{attribute 'linkalways'} 
{attribute 'no_explicit_call' := 'This FB is a CLASS and must be accessed using methods or properties'}
{attribute 'enable_dynamic_creation'}
FUNCTION_BLOCK FINAL MAX_UDINT EXTENDS Node
VAR
	in1 : _UDINT(0);
	in2 : _UDINT(0);
	out : _UDINT(0);
END_VAR

METHOD PUBLIC Clone : I_Node
VAR
	pNode : POINTER TO MAX_UDINT;
END_VAR
pNode := __NEW(MAX_UDINT);
Clone := pNode^;
END_METHOD

METHOD FB_init : BOOL
VAR_INPUT
	bInitRetains : BOOL; // if TRUE, the retain variables are initialized (warm start / cold start)
	bInCopyCode : BOOL;  // if TRUE, the instance afterwards gets moved into the copy code (online change)
END_VAR
AddInput('in1',THIS^.in1);
AddInput('in2',THIS^.in2);
AddOutput('out', THIS^.out);
END_METHOD

METHOD PROTECTED OnExecute
VAR
END_VAR
out.Value := MAX(in1.Value, in2.Value);
END_METHOD

END_FUNCTION_BLOCK

(* stored: Version 1.1.0.1, ProductVersion 3.1.4024.15
   POU MAX_UDINT: Id {2e8387af-4722-43a4-a1e9-55e7a16c698f}, SpecialFunc None
   Folder Constructor: Id {a89d2098-e33d-4e3d-9c8f-6a23b2150f97}
   Method Clone: Id {d1831383-fa73-491a-a42f-b34112e1b601}
   Method FB_init: Id {65915ac0-de7d-48fc-bf18-823ff2bcc712}
   Method OnExecute: Id {0d02a9e5-fe62-403f-8d3e-a6b629b312ea} *)
